PROGRAM BackgroundSerialCtrl
VAR
	fbUSBCtrl		: SerialLineControlADS;
	stComSerialCfg	: ComSerialConfig;
END_VAR

stComSerialCfg.Baudrate := 9600;
stComSerialCfg.ComPort := 3;
stComSerialCfg.DataBits := 8;
stComSerialCfg.StopBits := Tc2_SerialCom.STOPBITS_ONE;
stComSerialCfg.Parity := Tc2_SerialCom.PARITY_NONE;

fbUSBCtrl(
	Connect:= TRUE, 
	SerialCfg:= stComSerialCfg, 
	NetId:= '', 
	Timeout:= T#1S, 
	TxBuffer:= TxBuffer, 
	RxBuffer:= RxBuffer, 
	PortOpened=> , 
	Error=> , 
	ErrorID=> , 
	Busy=> , 
	TxBufCount=> , 
	RxBufCount=> );

END_PROGRAM

(* stored: Version 1.1.0.1, ProductVersion 3.1.4024.14
   POU BackgroundSerialCtrl: Id {de849666-5409-4aee-9afa-b79b122a0fcb}, SpecialFunc None *)
